RoboDK station: Dexter.rdk

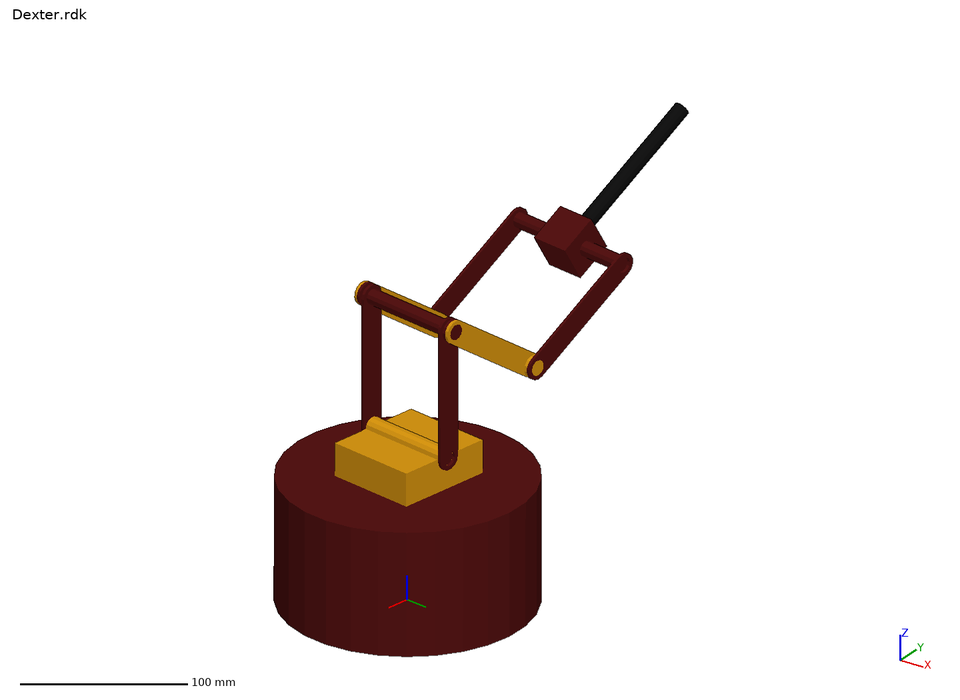
[picture v0: the station drawn from its stored meshes, robots at their saved joint values, targets as dots, program paths as lines]
Station Dexter (saved by RoboDK 5.9.6). Poses are relative to the parent item; angles as X-Y-Z fixed-axis rotations.
  - frame Frame 1 at (-0.78, -0.88, -0.95) mm, rotated rx 0.33 ry -0.82 rz -98.45 deg
  - object ER2_Fusion at (0, 0, 0) mm, geometry from ER2_Fusion.step
    - object Link_1 at (-0.36, -0.68, 0) mm, rotated rx 0 ry -0.14 rz -98.83 deg, size 159.5 x 159.8 x 82 mm
    - object Link_2 at (0, 0, 0) mm, size 73.3 x 110.6 x 122.9 mm
    - object Link_3 at (0, 0, 0) mm, size 78.6 x 27 x 100.8 mm
    - object Link_4 at (0, 0, 0) mm, size 95.4 x 90.9 x 58.6 mm
    - object Link_5 at (0, 0, 0) mm, size 103.4 x 106.8 x 68.2 mm
    - object Link_6 at (0, 0, 0) mm, size 23.7 x 87.7 x 57.6 mm
